// TwinCAT 3 PLC project Project_P1
// Title: Standard_Tools
// Company: MyCompany AB
// Author: Gulyawar Aman
// ProjectVersion: 0.1.0.0
// Description: This block tracks how many times a machine part has cycled and triggers a maintenance alarm when it hits a limit. It is ideal for a library because it is a generic tool we can reuse in many different projects.
// ProgramVersion: 3.1.4024.0
// libraries:
//   Tc2_Standard, * (Beckhoff Automation GmbH)
//   Tc2_System, * (Beckhoff Automation GmbH)
//   Tc3_Module, * (Beckhoff Automation GmbH)
// project tree:
//   / PlcTask.TcTTO
//   POUs/ FB_MaintenanceCounter.TcPOU
//   Version/ Global_Version.TcGVL
// real-time tasks:
//   TASK PlcTask: cycle T#10ms, priority 20, ADS port 350

CONFIGURATION Project_P1
    RESOURCE PLC ON TwinCAT3
        TASK PlcTask(INTERVAL := T#10ms, PRIORITY := 20);
        PROGRAM MAIN WITH PlcTask : MAIN;
    END_RESOURCE
END_CONFIGURATION

// ---- Version/Global_Version.TcGVL
{attribute 'TcGenerated'}
{attribute 'no-analysis'}
{attribute 'linkalways'}
// This function has been automatically generated from the project information.
VAR_GLOBAL CONSTANT
	{attribute 'const_non_replaced'}
	stLibVersion_Standard_Tools : ST_LibVersion := (iMajor := 0, iMinor := 1, iBuild := 0, iRevision := 0, nFlags := 0, sVersion := '0.1.0.0');
END_VAR

// ---- POUs/FB_MaintenanceCounter.TcPOU
FUNCTION_BLOCK FB_MaintenanceCounter
VAR_INPUT
    bCountPulse      : BOOL;   
    bReset           : BOOL;   
    nLimit           : UDINT;  
END_VAR
VAR_OUTPUT
    nCurrentCount    : UDINT;  
    bMaintenanceDue  : BOOL;   
END_VAR
VAR
    fbRisingEdge     : R_TRIG; 
END_VAR


fbRisingEdge(CLK := bCountPulse);


IF fbRisingEdge.Q THEN
    nCurrentCount := nCurrentCount + 1;
END_IF

IF bReset THEN
    nCurrentCount := 0;
END_IF


bMaintenanceDue := (nCurrentCount >= nLimit) AND (nLimit > 0);

END_FUNCTION_BLOCK
